// TIA Portal V15.1 export
// export: Created 2020-06-12T07:15:58.9726562Z, ExportSetting None, DisplayName Totally Integrated Automation Portal, DisplayVersion V15.1, DisplayName TIA Portal Openness, DisplayVersion V15.1, DisplayName STEP 7 Professional, DisplayVersion V15.1, DisplayName STEP 7 Safety, DisplayVersion V15.1, DisplayName WinCC Advanced, DisplayVersion V15.1
DATA_BLOCK "ai"   // DB2
{ S7_Optimized_Access := 'TRUE' }
AUTHOR : atec_osm
FAMILY : COMMON
NAME : AnaVal
VERSION : 2.0
// stored: MemoryReserve 100
   VAR
      ES1LD1_CV01 { ExternalAccessible := 'False'; ExternalVisible := 'False'; ExternalWritable := 'False'} : Real := 0.4340278;   // Control Valve Dedusting System Actual Value
      ES1LV1_PT01 { ExternalAccessible := 'False'; ExternalVisible := 'False'; ExternalWritable := 'False'} : Real := 0.0;   // Pressure Transmitter MPS FL
      ES1LT1_XT01_volt { ExternalAccessible := 'False'; ExternalVisible := 'False'; ExternalWritable := 'False'} : Real := 0.07559317;   // Actual voltage transducer
      ES1LT1_XT01_pwr { ExternalAccessible := 'False'; ExternalVisible := 'False'; ExternalWritable := 'False'} : Real := 0.0;   // Actual power transducer
      ES1LT1_XT01_cur { ExternalAccessible := 'False'; ExternalVisible := 'False'; ExternalWritable := 'False'} : Real := 0.01446759;   // Actual current transducer
      ES1LT1_QT01 { ExternalAccessible := 'False'; ExternalVisible := 'False'; ExternalWritable := 'False'} : Real := 0.0;   // Earth Leakage Current
      ES1LV1_PT02 { ExternalAccessible := 'False'; ExternalVisible := 'False'; ExternalWritable := 'False'} : Real := 0.0;   // Pressure Transmitter MPS RL
      ES1LT1_XS01_temp1 { ExternalAccessible := 'False'; ExternalVisible := 'False'; ExternalWritable := 'False'} : Real := 0.0;   // Transformer Actual Temperatur Coil U
      ES1LT1_XS01_temp2 { ExternalAccessible := 'False'; ExternalVisible := 'False'; ExternalWritable := 'False'} : Real := 0.0;   // Transformer Actual Temperatur Coil V
      ES1LT1_XS01_temp3 { ExternalAccessible := 'False'; ExternalVisible := 'False'; ExternalWritable := 'False'} : Real := 0.0;   // Transformer Actual Temperatur Coil W
      ES1LA2_PT01 { ExternalAccessible := 'False'; ExternalVisible := 'False'; ExternalWritable := 'False'} : Real := 0.0;   // Pressure Transmitter Sluice Alloy Addion Actual value
      ES1LE2_M01pos { ExternalAccessible := 'False'; ExternalVisible := 'False'; ExternalWritable := 'False'} : Real := 3.011068;   // X-Adjustment Actual position
      ES1LE2_M02pos { ExternalAccessible := 'False'; ExternalVisible := 'False'; ExternalWritable := 'False'} : Real := 9.103733;   // Y-Adjustment Actual position
      ES1LC3_TT02 { ExternalAccessible := 'False'; ExternalVisible := 'False'; ExternalWritable := 'False'} : Real := 35.42028;   // Temperature Transmitter Power Ram Outer Pipe RL Actual value
      ES1LC3_TT04 { ExternalAccessible := 'False'; ExternalVisible := 'False'; ExternalWritable := 'False'} : Real := 35.32263;   // TT Conduction Rail 1+2 RL Actual value
      ES1LC3_TT06 { ExternalAccessible := 'False'; ExternalVisible := 'False'; ExternalWritable := 'False'} : Real := 35.03689;   // Temperature Transmitter Gas Hood RL Actual value
      ES1LE2_XT01 { ExternalAccessible := 'False'; ExternalVisible := 'False'; ExternalWritable := 'False'} : Real := 0.0;   // Actual Voltage Power Ram
      ES1LE3_PT01 { ExternalAccessible := 'False'; ExternalVisible := 'False'; ExternalWritable := 'False'} : Real := 5000.0;   // Pressure Transmitter Protective Gas Hood 1 Actual value
      ES1LE3_PT02 { ExternalAccessible := 'False'; ExternalVisible := 'False'; ExternalWritable := 'False'} : Real := 0.8289928;   // Pressure Transmitter Protective Gas Hood 2 Actual value
      ES1LE3_QT01_O2 { ExternalAccessible := 'False'; ExternalVisible := 'False'; ExternalWritable := 'False'} : Real := 16.27732;   // Oxygen Measurement System
      ES1LE3_QT01_O2hw { ExternalAccessible := 'False'; ExternalVisible := 'False'; ExternalWritable := 'False'} : Real := 0.0;   // Oxygen Measurement System
      ES1LE3_XT01 { ExternalAccessible := 'False'; ExternalVisible := 'False'; ExternalWritable := 'False'} : Real := 0.001808449;   // Current Measuring Hood RL 1 act current
      ES1LE3_XT02 { ExternalAccessible := 'False'; ExternalVisible := 'False'; ExternalWritable := 'False'} : Real := 0.002893519;   // Current Measuring Hood RL 2 act current
      ES1LE3_XT03 { ExternalAccessible := 'False'; ExternalVisible := 'False'; ExternalWritable := 'False'} : Real := 0.004340278;   // Current Measuring Hood RL 3 act current
      ES1LE3_XT04 { ExternalAccessible := 'False'; ExternalVisible := 'False'; ExternalWritable := 'False'} : Real := 0.004340278;   // Current Measuring Hood RL 4 act current
      ES1LZ1_PT01 { ExternalAccessible := 'False'; ExternalVisible := 'False'; ExternalWritable := 'False'} : Real := 998.1193;   // Pressure Transmitter Atmosphere
      ES1LC1_CV01 { ExternalAccessible := 'False'; ExternalVisible := 'False'; ExternalWritable := 'False'} : Real := 90.39714;   // Actual value Control valve RL Heat Exchanger
      ES1LC1_PT01 { ExternalAccessible := 'False'; ExternalVisible := 'False'; ExternalWritable := 'False'} : Real := 4.021122;   // Foreward Line Strainer Pressure Actual value
      ES1LC1_PT02 { ExternalAccessible := 'False'; ExternalVisible := 'False'; ExternalWritable := 'False'} : Real := 3.932292;   // Return Line Strainer Pressure Actual value
      ES1LC1_dP02 { ExternalAccessible := 'False'; ExternalVisible := 'False'; ExternalWritable := 'False'} : Real := 0.08883071;   // Differential pressure strainer
      ES1LC1_PT03 { ExternalAccessible := 'False'; ExternalVisible := 'False'; ExternalWritable := 'False'} : Real := 0.142636;   // Pressure Transmitter CW Tank
      ES1LC1_QT01 { ExternalAccessible := 'False'; ExternalVisible := 'False'; ExternalWritable := 'False'} : Real := 28.39265;   // CW Tank actual conductivity
      ES1LC1_TT01 { ExternalAccessible := 'False'; ExternalVisible := 'False'; ExternalWritable := 'False'} : Real := 27.74523;   // CW Tank Temperature Actual value
      ES1LC1_TT02 { ExternalAccessible := 'False'; ExternalVisible := 'False'; ExternalWritable := 'False'} : Real := 25.96571;   // Temperature Transmitter CW Recooling HE FL Actual value
      ES1LC1_TT03 { ExternalAccessible := 'False'; ExternalVisible := 'False'; ExternalWritable := 'False'} : Real := 28.54456;   // Temperature Transmitter CW Recooling HE RL Actual value
      ES1LC1_TT04 { ExternalAccessible := 'False'; ExternalVisible := 'False'; ExternalWritable := 'False'} : Real := 28.51201;   // Temperature Transmitter CW HE FL Actual value
      ES1LC3_TT01 { ExternalAccessible := 'False'; ExternalVisible := 'False'; ExternalWritable := 'False'} : Real := 31.20298;   // TT Electrode Column RL Actual value
      ES1LC5_CV01 { ExternalAccessible := 'False'; ExternalVisible := 'False'; ExternalWritable := 'False'} : Real := 0.0;   // Actual value Control Valve CW Melt Station 1 RL
      ES1LC5_CV02 { ExternalAccessible := 'False'; ExternalVisible := 'False'; ExternalWritable := 'False'} : Real := 24.86979;   // Actual value Control Valve CW Baseplate 1 RL
      ES1LC5_FT01 { ExternalAccessible := 'False'; ExternalVisible := 'False'; ExternalWritable := 'False'} : Real := 0.01808449;   // Flow Transmitter CW Static Mould MS1 RL Actual value
      ES1LC5_FT02 { ExternalAccessible := 'False'; ExternalVisible := 'False'; ExternalWritable := 'False'} : Real := 0.0;   // Flow Transmitter CW Baseplate MS1 RL Actual value
      ES1LC5_PT01 { ExternalAccessible := 'False'; ExternalVisible := 'False'; ExternalWritable := 'False'} : Real := 0.2583912;   // Pressure Transmitter CW Melt Station 1 RL Actual value
      ES1LC5_PT02 { ExternalAccessible := 'False'; ExternalVisible := 'False'; ExternalWritable := 'False'} : Real := 0.2690972;   // Pressure Transmitter CW Baseplate 1 RL value
      ES1LC5_TT01 { ExternalAccessible := 'False'; ExternalVisible := 'False'; ExternalWritable := 'False'} : Real := 27.81756;   // Temperature Transmitter CW Melt Station 1+2 FL Actual value
      ES1LC5_TT02 { ExternalAccessible := 'False'; ExternalVisible := 'False'; ExternalWritable := 'False'} : Real := 24.4647;   // TT CW Static Mould MS1 RL Actual value
      ES1LC5_TT04 { ExternalAccessible := 'False'; ExternalVisible := 'False'; ExternalWritable := 'False'} : Real := 23.22049;   // Temperature Transmitter CW Baseplate 1 RL Actual value
      ES1LC5_TT07 { ExternalAccessible := 'False'; ExternalVisible := 'False'; ExternalWritable := 'False'} : Real := 26.63845;   // TT Baseplate Clamp MS1 RL Actual value
      ES1LC5_TT08 { ExternalAccessible := 'False'; ExternalVisible := 'False'; ExternalWritable := 'False'} : Real := 26.89887;   // TT Current Pipes MS1 RL Actual value
      ES1LC6_CV01 { ExternalAccessible := 'False'; ExternalVisible := 'False'; ExternalWritable := 'False'} : Real := 12.68446;   // Actual value Control Valve CW Melt Station 2 RL
      ES1LC6_CV02 { ExternalAccessible := 'False'; ExternalVisible := 'False'; ExternalWritable := 'False'} : Real := 0.0;   // Actual value Control Valve CW Baseplate 2 RL
      ES1LC6_FT01 { ExternalAccessible := 'False'; ExternalVisible := 'False'; ExternalWritable := 'False'} : Real := 19.81698;   // Flow Transmitter CW Static Mould MS2 RL Actual value
      ES1LC6_FT02 { ExternalAccessible := 'False'; ExternalVisible := 'False'; ExternalWritable := 'False'} : Real := 12.2092;   // Flow Transmitter CW Baseplate 2 RL Actual value
      ES1LC6_PT01 { ExternalAccessible := 'False'; ExternalVisible := 'False'; ExternalWritable := 'False'} : Real := 2.757234;   // Pressure Transmitter CW Melt Station 2 RL Actual value
      ES1LC6_PT02 { ExternalAccessible := 'False'; ExternalVisible := 'False'; ExternalWritable := 'False'} : Real := 0.9088542;   // Pressure Transmitter CW Baseplate 2 RL value
      ES1LC6_TT02 { ExternalAccessible := 'False'; ExternalVisible := 'False'; ExternalWritable := 'False'} : Real := 28.67477;   // Temperature Transmitter CW Static Mould MS2 RL Actual value
      ES1LC6_TT04 { ExternalAccessible := 'False'; ExternalVisible := 'False'; ExternalWritable := 'False'} : Real := 25.78125;   // Temperature Transmitter CW Baseplate 2 RL Actual value
      ES1LC6_TT07 { ExternalAccessible := 'False'; ExternalVisible := 'False'; ExternalWritable := 'False'} : Real := 33.60098;   // TT Baseplate Clamp MS2 RL Actual value
      ES1LC6_TT08 { ExternalAccessible := 'False'; ExternalVisible := 'False'; ExternalWritable := 'False'} : Real := 31.83594;   // TT Current Pipes MS2 RL Actual value
      ES1LC7_CV01 { ExternalAccessible := 'False'; ExternalVisible := 'False'; ExternalWritable := 'False'} : Real := 80.30238;   // Actual value Control Valve CW Module Recooling HE RL
      ES1LC7_PT10 { ExternalAccessible := 'False'; ExternalVisible := 'False'; ExternalWritable := 'False'} : Real := 1.918113;   // Pressure Transmitter CW Module Pump FL Actual value
      ES1LC7_TT01 { ExternalAccessible := 'False'; ExternalVisible := 'False'; ExternalWritable := 'False'} : Real := 34.69329;   // Temperature Transmitter CW Transductor RL Actual value
      ES1LC7_TT02 { ExternalAccessible := 'False'; ExternalVisible := 'False'; ExternalWritable := 'False'} : Real := 34.11097;   // TT CW Current Condution F&amp;B RL Actual value
      ES1LC7_TT10 { ExternalAccessible := 'False'; ExternalVisible := 'False'; ExternalWritable := 'False'} : Real := 33.26823;   // Temperature Transmitter CW Module Pump FL Actual value
      ES1LC7_TT12 { ExternalAccessible := 'False'; ExternalVisible := 'False'; ExternalWritable := 'False'} : Real := 35.43837;   // Temperature Transmitter CW Module HE FL Actual value
      ES1LC7_TT13 { ExternalAccessible := 'False'; ExternalVisible := 'False'; ExternalWritable := 'False'} : Real := 33.70226;   // Temperature Transmitter CW Module HE RL Actual value
      ES1LC7_TT14 { ExternalAccessible := 'False'; ExternalVisible := 'False'; ExternalWritable := 'False'} : Real := 34.76924;   // TT CW Module Recooling HE RL Actual value
      ES1LC7_TT15 { ExternalAccessible := 'False'; ExternalVisible := 'False'; ExternalWritable := 'False'} : Real := 26.20081;   // TT CW Module Recooling HE FL Actual value
      ES1LC7_TT16 { ExternalAccessible := 'False'; ExternalVisible := 'False'; ExternalWritable := 'False'} : Real := 11.25;   // TT CW Vacuum Dry Screw Pump RL Actual value
      ES1LC7_TT17 { ExternalAccessible := 'False'; ExternalVisible := 'False'; ExternalWritable := 'False'} : Real := 0.0;   // TT CW Vacuum Roots Pump RL Actual value
      ES1LC9_QT01 { ExternalAccessible := 'False'; ExternalVisible := 'False'; ExternalWritable := 'False'} : Real := 0.0;
      ES1LC9_TT01 { ExternalAccessible := 'False'; ExternalVisible := 'False'; ExternalWritable := 'False'} : Real := 25.22787;
      ES1LC9_FT01 { ExternalAccessible := 'False'; ExternalVisible := 'False'; ExternalWritable := 'False'} : Real := 15.78993;
      ES1LC9_FT02 { ExternalAccessible := 'False'; ExternalVisible := 'False'; ExternalWritable := 'False'} : Real := 4.954789;
      ES1LC9_PT01 { ExternalAccessible := 'False'; ExternalVisible := 'False'; ExternalWritable := 'False'} : Real := 3.00897;
      ES1LG1_CV01 { ExternalAccessible := 'False'; ExternalVisible := 'False'; ExternalWritable := 'False'} : Real := 0.0;   // Control Valve Ar PGH Act Flow
      ES1LG1_CV02 { ExternalAccessible := 'False'; ExternalVisible := 'False'; ExternalWritable := 'False'} : Real := 80.0;   // Control Valve N2 PGH Act Flow
      AX1LD3_PT01 { ExternalAccessible := 'False'; ExternalVisible := 'False'; ExternalWritable := 'False'} : Real := 3.338397;   // Dedusting line pressure
      AX1LD3_PT02 { ExternalAccessible := 'False'; ExternalVisible := 'False'; ExternalWritable := 'False'} : Real := 1.215277;   // Dedusting filter pressure
   END_VAR
BEGIN
END_DATA_BLOCK
